(* PLC project Unnamed, Unknown Unnamed 1 *)
(* stored: creationDateTime 2026-02-02T17:47:50, modificationDateTime 2026-02-02T17:55:39 *)

PROGRAM program0
  VAR
    PillSensorA AT %I0.3 : BOOL;
    PillSensorB AT %I0.5 : BOOL;
    ResetAlarm AT %I0.6 : BOOL;
    Alarm AT %M03 : BOOL;
  END_VAR
  VAR
    CTU0 : CTU;
    ErrorCount : INT;
    Error : BOOL;
  END_VAR
  VAR  (* added by the conversion: wires and edge detectors of the diagram *)
    R_TRIG1 : R_TRIG;
    R_TRIG2 : R_TRIG;
  END_VAR

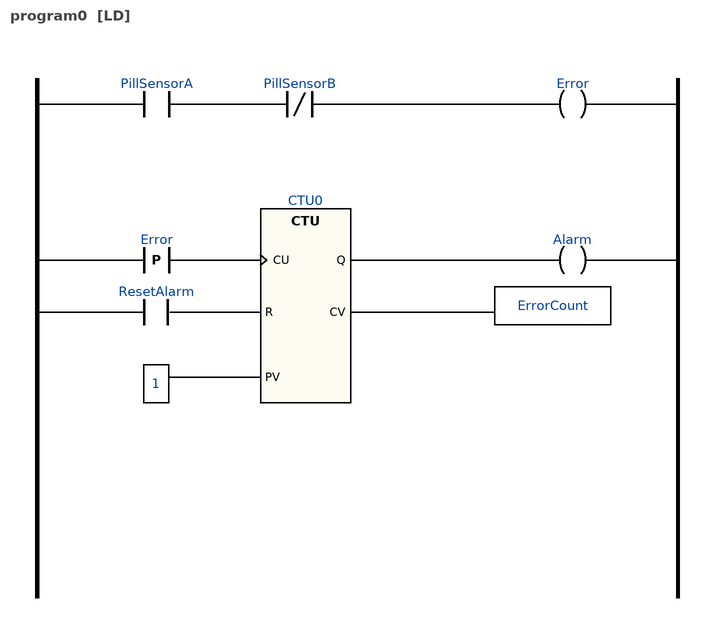
(* LD diagram, written out as Structured Text *)
Error := PillSensorA AND NOT PillSensorB;
R_TRIG1(CLK := Error);
R_TRIG2(CLK := R_TRIG1.Q);
CTU0(CU := R_TRIG2.Q, R := ResetAlarm, PV := 1);
ErrorCount := CTU0.CV;
Alarm := CTU0.Q;
END_PROGRAM

CONFIGURATION Config0
  RESOURCE Res0 ON PLC
    TASK task0(INTERVAL := T#20ms, PRIORITY := 0);
    PROGRAM instance0 WITH task0 : program0;
  END_RESOURCE
END_CONFIGURATION
